(* Logix 5000 project; controller Carpenter_Meter_SCP vendor 1 type 14 code 217 rev 31.11; software revision 31.01; part 7 of 7 *)
(* tags used below, declared in another part *)
   alarm_co : BOOL[32];
   Alarm_horn_req : BOOL;   // Alarm Horn Request
   Carpenter_to_Pawnee_OK : BOOL;   // Carpenter to Pawnee Flow Path Permissive
   Cust1_WIOM_Alarm : BOOL;   // Customer 1 WIOM Alarm
   ovrd_esd : Override;   // ESD Override
   Sta_Stat : StaStatus;
   valve_failure : BOOL;   // Valve Failure Override
   valve_SD_tmr : TIMER;   // Valve Failure Station Stop Timer
   XV_0001 : BaseVLVLiquid;   // XV-0001
   XV_0001_AOI : Valve_Control;   // XV-0001 Control
   XV_0041 : BaseVLVLiquid;   // XV-0041
   XV_0041_AOI : Valve_Control;   // XV-0041 Control
   XV_1100 : BaseVLVLiquid;   // XV-1100
   XV_1100_AOI : Valve_Control;   // XV-1100 Control
   XV_1101 : BaseVLVLiquid;   // XV-1101
   XV_1101_AOI : Valve_Control;   // XV-1100 Control
(* Station_Overrides, continued *)

ROUTINE Valve_Failure   (* ladder *)
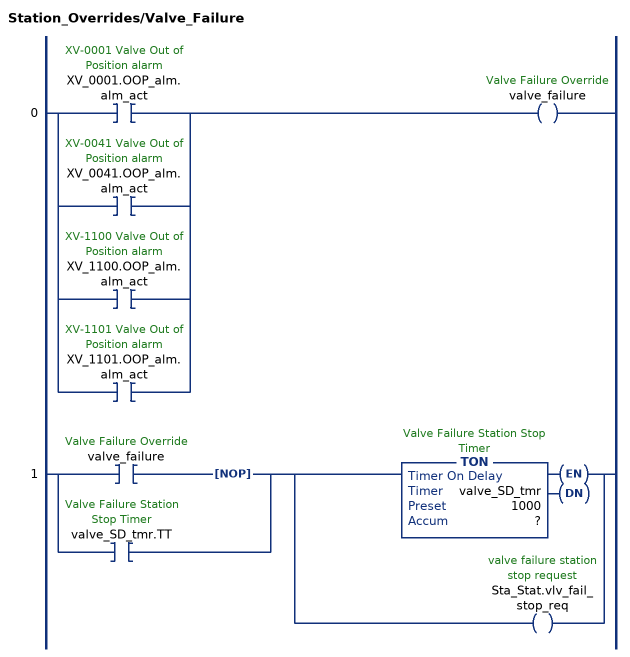
   0: [XIC(XV_0001.OOP_alm.alm_act) ,XIC(XV_0041.OOP_alm.alm_act) ,XIC(XV_1100.OOP_alm.alm_act) ,XIC(XV_1101.OOP_alm.alm_act) ]OTE(valve_failure);
   1: [XIC(valve_failure) NOP() ,XIC(valve_SD_tmr.TT) ][TON(valve_SD_tmr,?,?) ,OTE(Sta_Stat.vlv_fail_stop_req) ];
END_ROUTINE
END_PROGRAM

PROGRAM Valve_Control   (* main routine Station_Valves *)

ROUTINE Station_Valves   (* ladder *)
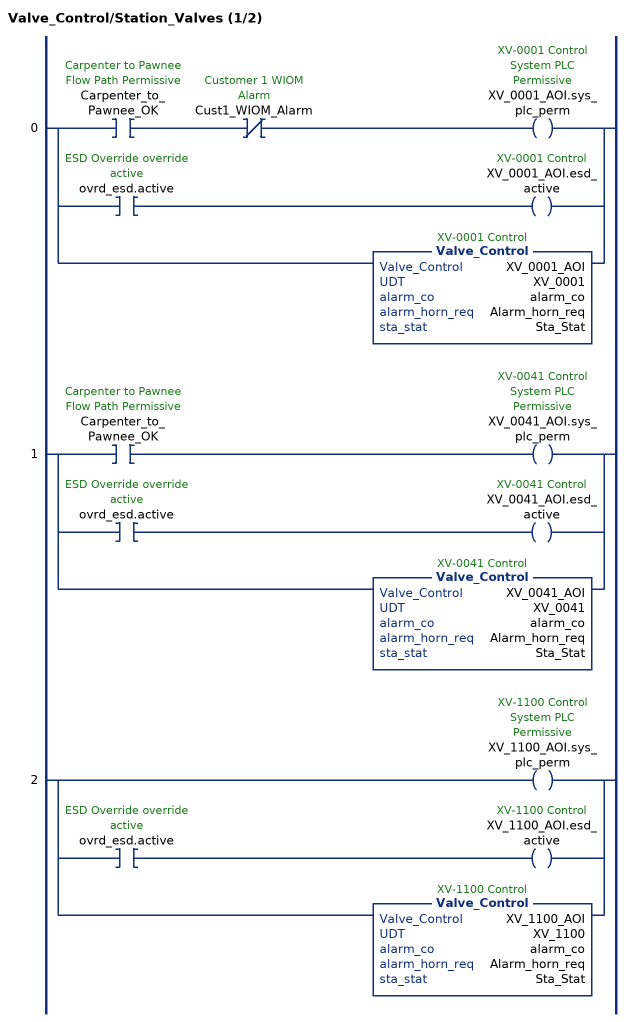
   0: [XIC(Carpenter_to_Pawnee_OK) XIO(Cust1_WIOM_Alarm) OTE(XV_0001_AOI.sys_plc_perm) ,XIC(ovrd_esd.active) OTE(XV_0001_AOI.esd_active) ,Valve_Control(XV_0001_AOI,XV_0001,alarm_co,Alarm_horn_req,Sta_Stat) ];
   1: [XIC(Carpenter_to_Pawnee_OK) OTE(XV_0041_AOI.sys_plc_perm) ,XIC(ovrd_esd.active) OTE(XV_0041_AOI.esd_active) ,Valve_Control(XV_0041_AOI,XV_0041,alarm_co,Alarm_horn_req,Sta_Stat) ];
   2: [OTE(XV_1100_AOI.sys_plc_perm) ,XIC(ovrd_esd.active) OTE(XV_1100_AOI.esd_active) ,Valve_Control(XV_1100_AOI,XV_1100,alarm_co,Alarm_horn_req,Sta_Stat) ];
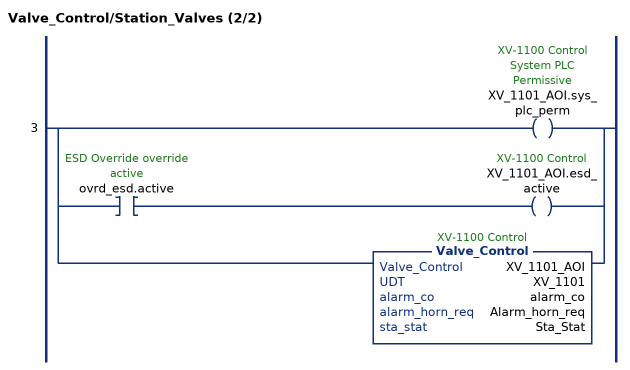
   3: [OTE(XV_1101_AOI.sys_plc_perm) ,XIC(ovrd_esd.active) OTE(XV_1101_AOI.esd_active) ,Valve_Control(XV_1101_AOI,XV_1101,alarm_co,Alarm_horn_req,Sta_Stat) ];
END_ROUTINE
END_PROGRAM
